SUBAPPLICATION Uebung_004b2 (* Toggle Flip-Flop mit IE / Split / doppelt *)
  (* Standard: 61499-2; Description: Copyright (c) 2023 Meisterschulen am Ostbahnhof This program and the accompanying materials are made available under the terms of the Eclipse Public License 2.0 which is available at https://www.eclipse.org/legal/epl-2.0/ SPDX-License-Identifier: EPL-2.0 *)
  (* Version 1.0, 2023-10-23, Franz Höpfinger, Meisterschulen am Ostbahnhof *)
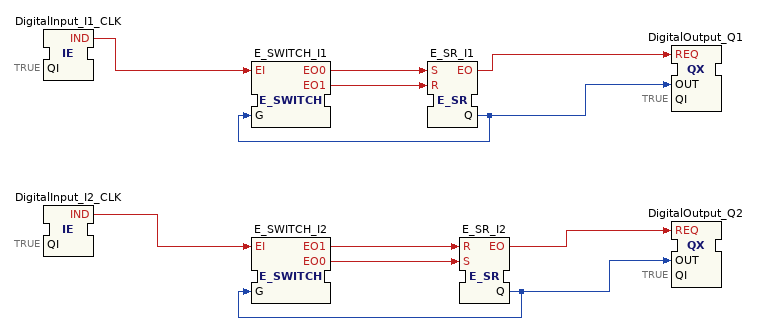
  FBS
    DigitalOutput_Q1 : QX(QI := TRUE);
    DigitalInput_I1_CLK : IE(QI := TRUE);
    E_SR_I1 : E_SR;
    E_SWITCH_I1 : E_SWITCH;
    E_SWITCH_I2 : E_SWITCH;
    DigitalOutput_Q2 : QX(QI := TRUE);
    E_SR_I2 : E_SR;
    DigitalInput_I2_CLK : IE(QI := TRUE);
  END_FBS
  EVENT_CONNECTIONS
    E_SR_I1.EO TO DigitalOutput_Q1.REQ;
    DigitalInput_I1_CLK.IND TO E_SWITCH_I1.EI;
    E_SWITCH_I1.EO0 TO E_SR_I1.S;
    E_SWITCH_I1.EO1 TO E_SR_I1.R;
    E_SWITCH_I2.EO1 TO E_SR_I2.R;
    E_SWITCH_I2.EO0 TO E_SR_I2.S;
    E_SR_I2.EO TO DigitalOutput_Q2.REQ;
    DigitalInput_I2_CLK.IND TO E_SWITCH_I2.EI;
  END_CONNECTIONS
  DATA_CONNECTIONS
    E_SR_I1.Q TO DigitalOutput_Q1.OUT;
    E_SR_I1.Q TO E_SWITCH_I1.G;
    E_SR_I2.Q TO E_SWITCH_I2.G;
    E_SR_I2.Q TO DigitalOutput_Q2.OUT;
  END_CONNECTIONS
END_SUBAPPLICATION
